# EPICS IOC start-up script: iocsh/Oxford_ILM202.iocsh
# ### Oxford_ILM202.iocsh ###

#- ###################################################
#- PREFIX         - IOC Prefix
#- INSTANCE       - Instance Prefix
#- PORT           - Serial port name
#- IP             - Location of IP module
#- ###################################################

#- Oxford ILM202 Cryogen Level Meter
asynSetOption("$(PORT)", -1, "baud",    "9600")
asynSetOption("$(PORT)", -1, "bits",    "8")
asynSetOption("$(PORT)", -1, "stop",    "1")
asynSetOption("$(PORT)", -1, "parity",  "none")
asynSetOption("$(PORT)", -1, "clocal",  "Y")
asynSetOption("$(PORT)", -1, "crtscts", "N")

asynOctetSetInputEos( "$(PORT)", -1, "")
asynOctetSetOutputEos("$(PORT)", -1, "")

dbLoadRecords("$(IP)/ipApp/Db/Oxford_ILM202.db", "P=$(PREFIX),S=$(INSTANCE),PORT=$(PORT)")
